PROGRAM progSCACntrl
VAR
	Enable : BOOL;
	SCA_04_0100 : fbSCA;
END_VAR

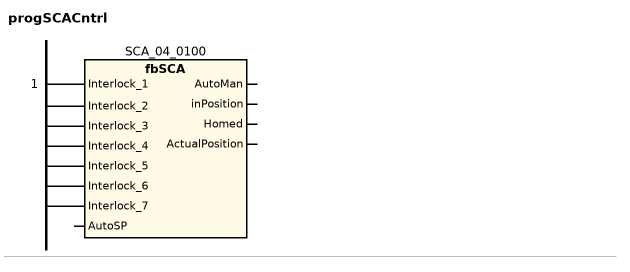
// NETWORK 1
SCA_04_0100(
    Interlock_1 := TRUE,
    Interlock_2 := TRUE,
    Interlock_3 := TRUE,
    Interlock_4 := TRUE,
    Interlock_5 := TRUE,
    Interlock_6 := TRUE,
    Interlock_7 := TRUE); // fbSCA

END_PROGRAM

(* stored: Version 1.1.0.1, ProductVersion 3.1.4022.17
   POU progSCACntrl: Id {137c8aef-24e8-40b2-a479-d60d1b8ced89}, SpecialFunc None *)
